FUNCTION_BLOCK ACTUORSbutton (* Basic Function Block Type *)
  (* Standard: 61499-2 *)
  (* Version 0.0, 05/07/2022, Etienne, Schneider Electric, Template *)
  PACKAGE Main;
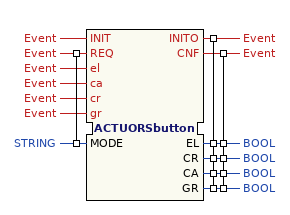
  EVENT_INPUT
    INIT; (* Initialization Request *)
    REQ WITH MODE;
    el; (* Normal Execution Request *)
    ca;
    cr;
    gr;
  END_EVENT
  EVENT_OUTPUT
    INITO WITH EL, CA, CR, GR; (* Initialization Confirm *)
    CNF WITH EL, CA, CR, GR; (* Execution Confirmation *)
  END_EVENT
  VAR_INPUT
    MODE : STRING;
  END_VAR
  VAR_OUTPUT
    EL : BOOL; (* Output event qualifier *)
    CR : BOOL;
    CA : BOOL;
    GR : BOOL;
  END_VAR
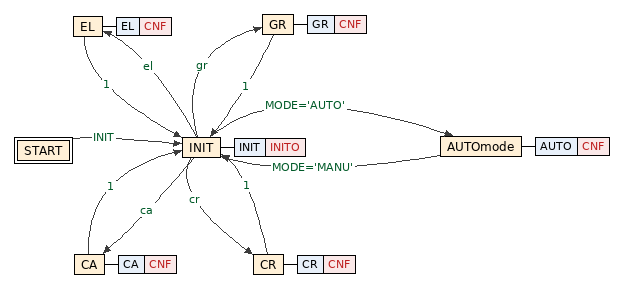
  EC_STATES
    START; (* Initial State *)
    INIT : INIT -> INITO; (* Initialization *)
    EL : EL -> CNF;
    CA : CA -> CNF;
    CR : CR -> CNF;
    GR : GR -> CNF;
    AUTOmode : AUTO -> CNF;
  END_STATES
  EC_TRANSITIONS
    START TO INIT := INIT;
    EL TO INIT := 1;
    GR TO INIT := 1;
    CA TO INIT := 1;
    CR TO INIT := 1;
    INIT TO EL := el;
    INIT TO GR := gr;
    INIT TO CA := ca;
    INIT TO CR := cr;
    INIT TO AUTOmode := MODE='AUTO';
    AUTOmode TO INIT := MODE='MANU';
  END_TRANSITIONS
  ALGORITHM INIT IN ST: (* Initialization algorithm *)
;
CA:=FALSE;
EL:=FALSE;
CR:=FALSE;
GR:=FALSE;
  END_ALGORITHM
  ALGORITHM EL IN ST: (* Normally executed algorithm *)
;
EL:=TRUE;
  END_ALGORITHM
  ALGORITHM CA IN ST:
;
CA:=TRUE;
  END_ALGORITHM
  ALGORITHM CR IN ST:
;
CR:=TRUE;
  END_ALGORITHM
  ALGORITHM GR IN ST:
;
GR:=TRUE;
  END_ALGORITHM
  ALGORITHM AUTO IN ST:
;
CA:=TRUE;
EL:=TRUE;
CR:=TRUE;
GR:=TRUE;
  END_ALGORITHM
END_FUNCTION_BLOCK
